// TIA Portal V18 export
TYPE "UDT_StopperInterface"
   STRUCT
      StopperRelease : Bool;
      StationReady : Bool;
      ProcessReady : Bool;
      Moving : Bool;
      Done : Bool;
      MissingError : Bool;
      ArrNextError : Bool;
      StopperStatus : Int;
   END_STRUCT;
END_TYPE
